(* CoDeSys 2.3 export: COUNT_CHAR.EXP *)

(* POU String/COUNT_CHAR, ST *)
FUNCTION COUNT_CHAR : INT
VAR_INPUT
	str : STRING(STRING_LENGTH);
	chr : BYTE;
END_VAR
VAR
	l: INT;
	pt : POINTER TO BYTE;
	pos: INT;
END_VAR


(*
version 1.1	29. mar. 2008
programmer 		kurt
tested by		hugo

COUNT_CHAR counts how often a character CHAR occurs within a string STR.

*)
PT := ADR(str);
l := LEN(str);
COUNT_CHAR := 0;
FOR pos := 1 TO l DO
	IF pt^ = CHR THEN COUNT_CHAR := COUNT_CHAR + 1; END_IF;
    PT := PT + 1;
END_FOR;


(* revision history
hm	29. feb 2008	rev 1.0
	original version

hm	29. mar. 2008	rev 1.1
	changed STRING to STRING(STRING_LENGTH)
*)
END_FUNCTION
